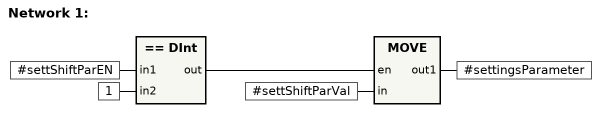
   IF #settShiftParEN = 1 THEN #settingsParameter := #settShiftParVal; END_IF;
END_REGION
END_FUNCTION

FUNCTION_BLOCK "wwwMain"   // FB9, FBD
{ S7_Optimized_Access := 'TRUE' }
VERSION : 0.1
// stored: AutoNumber true, IsIECCheckEnabled false, IsRetainMemResEnabled false, MemoryReserve 100, SetENOAutomatically false, UDAEnableTagReadback false
   VAR_TEMP
      RET_VAL : Int;
      temp : Int;
   END_VAR
BEGIN

REGION Network 1: ActualValues -> Web data
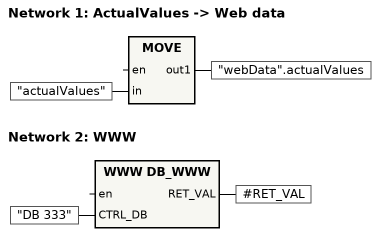
   "webData".actualValues := "actualValues";
END_REGION

REGION Network 2: WWW
   #RET_VAL := WWW(CTRL_DB := "DB 333");
END_REGION
END_FUNCTION_BLOCK

FUNCTION "outputConfig" : Void
{ S7_Optimized_Access := 'TRUE' }
VERSION : 0.1

BEGIN
	(*
	//Andon1
	"Andon1_greenLed" := "gDb_IO".Andon1.O_greenBtnLed;
	"Andon1_yellowLed" := "gDb_IO".Andon1.O_yellowBtnLed;
	"Andon1_redLed" := "gDb_IO".Andon1.O_redBtnLed;
	//Andon2
	"Andon2_greenLed" := "gDb_IO".Andon2.O_greenBtnLed;
	"Andon2_yellowLed" := "gDb_IO".Andon2.O_yellowBtnLed;
	"Andon2_redLed" := "gDb_IO".Andon2.O_redBtnLed;
	//Andon3
	"Andon3_greenLed" := "gDb_IO".Andon3.O_greenBtnLed;
	"Andon3_yellowLed" := "gDb_IO".Andon3.O_yellowBtnLed;
	"Andon3_redLed" := "gDb_IO".Andon3.O_redBtnLed;
	//Andon4
	"Andon4_greenLed" := "gDb_IO".Andon4.O_greenBtnLed;
	"Andon4_yellowLed" := "gDb_IO".Andon4.O_yellowBtnLed;
	"Andon4_redLed" := "gDb_IO".Andon4.O_redBtnLed;
	//Andon5
	"Andon5_greenLed" := "gDb_IO".Andon5.O_greenBtnLed;
	"Andon5_yellowLed" := "gDb_IO".Andon5.O_yellowBtnLed;
	"Andon5_redLed" := "gDb_IO".Andon5.O_redBtnLed;
	//Andon6
	"Andon6_greenLed" := "gDb_IO".Andon6.O_greenBtnLed;
	"Andon6_yellowLed" := "gDb_IO".Andon6.O_yellowBtnLed;
	"Andon6_redLed" := "gDb_IO".Andon6.O_redBtnLed;
	//Andon7
	"Andon7_greenLed" := "gDb_IO".Andon7.O_greenBtnLed;
	"Andon7_yellowLed" := "gDb_IO".Andon7.O_yellowBtnLed;
	"Andon7_redLed" := "gDb_IO".Andon7.O_redBtnLed;
	//Andon8
	"Andon8_greenLed" := "gDb_IO".Andon8.O_greenBtnLed;
	"Andon8_yellowLed" := "gDb_IO".Andon8.O_yellowBtnLed;
	"Andon8_redLed" := "gDb_IO".Andon8.O_redBtnLed;
	//Andon9
	"Andon9_greenLed" := "gDb_IO".Andon9.O_greenBtnLed;
	"Andon9_yellowLed" := "gDb_IO".Andon9.O_yellowBtnLed;
	"Andon9_redLed" := "gDb_IO".Andon9.O_redBtnLed;
	
	//SV1
	"SV1_green" := "gDb_IO".SignalColumn.O_green;
	"SV1_yellow" := "gDb_IO".SignalColumn.O_yellow;
	"SV1_red" := "gDb_IO".SignalColumn.O_red;
	
	//SV2
	"SV2_green" := "gDb_IO".SignalColumn.O_green;
	"SV2_yellow" := "gDb_IO".SignalColumn.O_yellow;
	"SV2_red" := "gDb_IO".SignalColumn.O_red;
	
	//Sirena
	"sir_start" := "gDb_IO".Sirene.O_sir_start;
	"sir_1" := "gDb_IO".Sirene.O_sirena_1;
	"sir_2" := "gDb_IO".Sirene.O_sirena_2;
	"sir_3" := "gDb_IO".Sirene.O_sirena_3;
	"sir_4" := "gDb_IO".Sirene.O_sirena_4;
	"sir_5" := "gDb_IO".Sirene.O_sirena_5;
	"sir_6" := "gDb_IO".Sirene.O_sirena_6;
	*)
END_FUNCTION

ORGANIZATION_BLOCK "Startup"
TITLE = "Complete Restart"
{ S7_Optimized_Access := 'TRUE' }
VERSION : 0.1

BEGIN
	// AndonBox enable
	"gDb_AndonBoxConfig".flashingPeriod := T#200ms;
	"gDb_AndonBoxConfig".EnableAndon1 := true;
	"gDb_AndonBoxConfig".EnableAndon2 := true;
	"gDb_AndonBoxConfig".EnableAndon3 := true;
	"gDb_AndonBoxConfig".EnableAndon4 := true;
	"gDb_AndonBoxConfig".EnableAndon5 := true;
	"gDb_AndonBoxConfig".EnableAndon6 := true;
	"gDb_AndonBoxConfig".EnableAndon7 := true;
	"gDb_AndonBoxConfig".EnableAndon8 := true;
	"gDb_AndonBoxConfig".EnableAndon9 := true;
	"gDb_AndonBoxConfig".EnableAndon10 := true;
	
	// Line name
	"webData".lineName := WSTRING#'LXX';
	
	// Andon text
	"webData".andon1Text := WSTRING#'Andon1';
	"webData".andon2Text := WSTRING#'Andon2';
	"webData".andon3Text := WSTRING#'Andon3';
	"webData".andon4Text := WSTRING#'Andon4';
	"webData".andon5Text := WSTRING#'Andon5';
	"webData".andon6Text := WSTRING#'Andon6';
	"webData".andon7Text := WSTRING#'Andon7';
	"webData".andon8Text := WSTRING#'Andon8';
	"webData".andon9Text := WSTRING#'Andon9';
	"webData".andon10Text := WSTRING#'Andon10';
	//test
END_ORGANIZATION_BLOCK

DATA_BLOCK "actualValues"   // DB21
{ S7_Optimized_Access := 'TRUE' }
VERSION : 0.1
// stored: AutoNumber true, DBAccessibleFromOPCUA true, DBAccessibleFromWebserver true, InstanceOfName UDT_actualValues, InstanceOfType UDT, IsOnlyStoredInLoadMemory false, IsWriteProtectedInAS false
"UDT_actualValues"
   // VAR RETAIN
   //    target { ExternalVisible := 'False'; ExternalWritable := 'False'} : DInt;
   //    actual { ExternalVisible := 'False'; ExternalWritable := 'False'} : DInt;
   //    ok { ExternalVisible := 'False'; ExternalWritable := 'False'} : DInt;
   //    difference { ExternalVisible := 'False'; ExternalWritable := 'False'} : DInt;
   //    counterTactTime { ExternalVisible := 'False'; ExternalWritable := 'False'} : DInt;
   //    state { ExternalVisible := 'False'; ExternalWritable := 'False'} : DInt;
   // END_VAR
BEGIN
END_DATA_BLOCK

DATA_BLOCK "control"   // DB6
{ S7_Optimized_Access := 'TRUE' }
// stored: InstanceOfName UDT_control, InstanceOfType UDT
"UDT_control"
   // VAR
   //    resetCounters { ExternalVisible := 'False'} : DInt;
   //    startTaktTimeCnt { ExternalVisible := 'False'} : DInt;
   //    stopTaktTimeCnt { ExternalVisible := 'False'} : DInt;
   //    actualMinus1 : DInt;
   //    actualPlus1 : DInt;
   //    okMinus1 : DInt;
   //    okPlus1 : DInt;
   // END_VAR
BEGIN
END_DATA_BLOCK

DATA_BLOCK "prePreviousValues"   // DB22
{ S7_Optimized_Access := 'TRUE' }
// stored: InstanceOfName UDT_actualValues, InstanceOfType UDT
"UDT_actualValues"
   // VAR RETAIN
   //    target { ExternalVisible := 'False'; ExternalWritable := 'False'} : DInt;
   //    actual { ExternalVisible := 'False'; ExternalWritable := 'False'} : DInt;
   //    ok { ExternalVisible := 'False'; ExternalWritable := 'False'} : DInt;
   //    difference { ExternalVisible := 'False'; ExternalWritable := 'False'} : DInt;
   //    counterTactTime { ExternalVisible := 'False'; ExternalWritable := 'False'} : DInt;
   //    state { ExternalVisible := 'False'; ExternalWritable := 'False'} : DInt;
   //    taktTime : DInt;
   // END_VAR
BEGIN
END_DATA_BLOCK

DATA_BLOCK "previousValues"   // DB19
{ S7_Optimized_Access := 'TRUE' }
VERSION : 0.1
// stored: AutoNumber true, DBAccessibleFromOPCUA true, DBAccessibleFromWebserver true, InstanceOfName UDT_actualValues, InstanceOfType UDT, IsOnlyStoredInLoadMemory false, IsWriteProtectedInAS false
"UDT_actualValues"
   // VAR RETAIN
   //    target { ExternalVisible := 'False'; ExternalWritable := 'False'} : DInt;
   //    actual { ExternalVisible := 'False'; ExternalWritable := 'False'} : DInt;
   //    ok { ExternalVisible := 'False'; ExternalWritable := 'False'} : DInt;
   //    difference { ExternalVisible := 'False'; ExternalWritable := 'False'} : DInt;
   //    counterTactTime { ExternalVisible := 'False'; ExternalWritable := 'False'} : DInt;
   //    state { ExternalVisible := 'False'; ExternalWritable := 'False'} : DInt;
   // END_VAR
BEGIN
END_DATA_BLOCK

DATA_BLOCK "settings"   // DB12
{ S7_Optimized_Access := 'TRUE' }
// stored: InstanceOfName UDT_settings, InstanceOfType UDT
"UDT_settings"
   // VAR RETAIN
   //    taktTimeCntOption { ExternalVisible := 'False'; S7_SetPoint := 'True'} : DInt;
   //    target { ExternalVisible := 'False'; S7_SetPoint := 'True'} : DInt;
   //    taktTime { ExternalVisible := 'False'; S7_SetPoint := 'True'} : DInt;
   //    countOption { ExternalVisible := 'False'; S7_SetPoint := 'True'} : DInt;
   // END_VAR
BEGIN
END_DATA_BLOCK

DATA_BLOCK "AndonMain_DB"   // DB5
VERSION : 0.1
// stored: AutoNumber true, DBAccessibleFromOPCUA true, DBAccessibleFromWebserver true, InstanceOfName AndonMain, InstanceOfType FB
"AndonMain"
BEGIN
END_DATA_BLOCK

DATA_BLOCK "nokButtonMain_DB"   // DB15
VERSION : 0.1
// stored: AutoNumber true, DBAccessibleFromOPCUA true, DBAccessibleFromWebserver true, InstanceOfName nokButtonMain, InstanceOfType FB
"nokButtonMain"
BEGIN
END_DATA_BLOCK

DATA_BLOCK "SireneMain_DB"   // DB10
VERSION : 0.1
// stored: AutoNumber true, DBAccessibleFromOPCUA true, DBAccessibleFromWebserver true, InstanceOfName SireneMain, InstanceOfType FB
"SireneMain"
BEGIN
END_DATA_BLOCK

DATA_BLOCK "wwwMain_DB"   // DB11
VERSION : 0.1
// stored: AutoNumber true, DBAccessibleFromOPCUA true, DBAccessibleFromWebserver true, InstanceOfName wwwMain, InstanceOfType FB
"wwwMain"
BEGIN
END_DATA_BLOCK

DATA_BLOCK "productionCounter_DB"   // DB18
VERSION : 0.1
// stored: AutoNumber true, DBAccessibleFromOPCUA true, DBAccessibleFromWebserver true, InstanceOfName productionCounter, InstanceOfType FB
"productionCounter"
BEGIN
END_DATA_BLOCK
